// TwinCAT 3 PLC project Example
// ProgramVersion: 3.1.4024.0
// libraries:
//   MTP, * (Zerlauth)
//   Tc2_MC2, * (Beckhoff Automation GmbH)
//   Tc2_Standard, * (Beckhoff Automation GmbH)
//   Tc2_System, * (Beckhoff Automation GmbH)
//   Tc2_Utilities, * (Beckhoff Automation GmbH)
//   Tc3_Module, * (Beckhoff Automation GmbH)
// project tree:
//   GVLs/ GVL.TcGVL
//   / plcTask1.TcTTO
//   POUs/Axis/ FB_McAxis.TcPOU, I_Axis.TcIO
//   POUs/ FB_Alarm.TcPOU, FB_Module01.TcPOU, MAIN.TcPOU
// real-time tasks:
//   TASK plcTask1: cycle T#1000ms, priority 20, ADS port 350

CONFIGURATION Example
    RESOURCE PLC ON TwinCAT3
        TASK plcTask1(INTERVAL := T#1000ms, PRIORITY := 20);
        PROGRAM Task1 WITH plcTask1 : Task1;
    END_RESOURCE
END_CONFIGURATION

// ---- GVLs/GVL.TcGVL
VAR_GLOBAL
	fbSaftey:		FB_Component;	
END_VAR

// ---- POUs/Axis/I_Axis.TcIO
INTERFACE I_Axis

END_INTERFACE

// ---- POUs/Axis/FB_McAxis.TcPOU
FUNCTION_BLOCK FB_McAxis EXTENDS FB_Component IMPLEMENTS I_Axis
VAR_INPUT
	bHome:				BOOL;
END_VAR
VAR_OUTPUT
END_VAR
VAR
	// Structs
	stAxis:							AXIS_REF;
	stParameter:					ST_AxisParameterSet;
	stComponents:					ST_AxisComponents;
	
	// General
	fbPower: 						MC_Power;
	fbReset: 						MC_Reset;
	fbHome: 						MC_Home;

	// Motion function blocks
	fbJog:							MC_Jog;
	fbSetPosition: 					MC_SetPosition;
	fbMoveAbsolute: 				REFERENCE TO MC_MoveAbsolute := fbMoveAbsolute1;
	fbMoveAbsolute1: 				MC_MoveAbsolute;
	fbMoveAbsolute2: 				MC_MoveAbsolute;
	fbMoveVelocity: 				MC_MoveVelocity;
	fbMoveRelative: 				MC_MoveRelative;
	fbHalt: 						MC_Halt;
	fbStop: 						MC_Stop;
	
	// Read function blocks
	fbReadAxisComponents:			MC_ReadAxisComponents;	
	fbReadError: 					MC_ReadAxisError;
	fbReadParameterSet:				MC_ReadParameterSet;	
	fbReadBoolParameter:			MC_ReadBoolParameter;
	fbReadParameter: 				MC_ReadParameter;
	
	// Write function blocks                            		
	fbWriteBoolParameter: 			MC_WriteBoolParameter;
	fbWriteBoolParameterPersistent: MC_WriteBoolParameterPersistent;
	fbWriteParameter: 				MC_WriteParameter;
	fbWriteParameterPersistent: 	MC_WriteParameterPersistent;
END_VAR
VAR PERSISTENT
	bCalibration:					BOOL;
	fHomePosition:					LREAL;
	fPositionCorrection:			LREAL;
	fMaximumForce:					LREAL;
END_VAR


SUPER^();

stAxis.ReadStatus();

fbPower(Axis:= stAxis);
	
fbReset(Axis:= stAxis);
fbReset.Execute:= FALSE;

fbJog(Axis:= stAxis);
fbJog.JogForward:= FALSE;
fbJog.JogBackwards:= FALSE;

fbHome(Axis:= stAxis);
fbHome.Execute:= FALSE;
	
fbSetPosition(Axis:= stAxis);
fbSetPosition.Execute:= FALSE;

fbMoveAbsolute1(Axis:= stAxis);
fbMoveAbsolute1.Execute:= FALSE;
	
fbMoveAbsolute2(Axis:= stAxis);
fbMoveAbsolute2.Execute:= FALSE;
	
fbMoveRelative(Axis:= stAxis);
fbMoveRelative.Execute:= FALSE;
	
fbMoveVelocity(Axis:= stAxis);
fbMoveVelocity.Execute:= FALSE;

fbHalt(Axis:= stAxis);
fbHalt.Execute:= FALSE;
	
fbStop(Axis:= stAxis);
fbStop.Execute:= FALSE;
	
fbReadBoolParameter(Axis:= stAxis);
fbReadBoolParameter.Enable:= FALSE;

fbWriteBoolParameter(Axis:= stAxis);
fbWriteBoolParameter.Execute:= FALSE;

fbWriteBoolParameterPersistent(Axis:= stAxis);
fbWriteBoolParameterPersistent.Execute:= FALSE;

fbReadParameter(Axis:= stAxis);
fbReadParameter.Enable:= FALSE;
	
fbWriteParameter(Axis:= stAxis);
fbWriteParameter.Execute:= FALSE;

fbWriteParameterPersistent(Axis:= stAxis);
fbWriteParameterPersistent.Execute:= FALSE;
	
fbReadParameterSet(Parameter:=stParameter, Axis:= stAxis);
fbReadParameterSet.Execute:= FALSE;

fbReadAxisComponents(AxisComponents:= stComponents, Axis:= stAxis);
fbReadError(Axis:= stAxis, Enable:= TRUE);

IF stAxis.Status.NcApplicationRequest THEN
	M_Home(stParameter.fEncRefPosition, MC_HomingMode.MC_Direct, TRUE);
END_IF

stAxis.PlcToNc.PositionCorrection:= fPositionCorrection;

METHOD M_Calibration : BOOL
VAR_INPUT
	fPrePosition:	LREAL;
	fPosition:		LREAL;
	fForce:			LREAL;
	fLimit:			LREAL;
	bEvaluation:	BOOL;
END_VAR
VAR_OUTPUT
	fDeviation:		LREAL;
END_VAR
END_METHOD

METHOD PUBLIC M_Halt : BOOL
VAR_INPUT
END_VAR
fbHalt.Execute:= TRUE;
M_Halt:= stAxis.Status.NotMoving;
END_METHOD

METHOD PUBLIC M_Home : BOOL
VAR_INPUT
	fPosition:					LREAL;
	eHomingMode:				MC_HomingMode;
	bClearPositionLag: 			BOOL;
END_VAR
fbHome.Execute:= TRUE;
fbHome.Position:= fPosition;
fbHome.HomingMode:= eHomingMode;
fbHome.Options.ClearPositionLag:= bClearPositionLag;
IF fbHome.Done THEN
	fbReset.Execute:= TRUE;
	M_Home:= TRUE;
END_IF
END_METHOD

METHOD PUBLIC M_Jog : BOOL
VAR_INPUT
	bPositive:	BOOL;
	bNegative:	BOOL;
	eMode:		E_JogMode;
END_VAR
fbJog.Mode:= eMode;
IF bPositive AND NOT bNegative THEN
	fbJog.JogForward:= TRUE;
ELSIF bNegative AND NOT bPositive THEN
	fbJog.JogBackwards:= TRUE;
END_IF
M_Jog:= fbJog.Active;
END_METHOD

METHOD PUBLIC M_MoveAbsolute : BOOL
VAR_INPUT
	fPosition:				LREAL;
	fVelocity:				LREAL;
	fAcceleration:			LREAL;
	fDeceleration:			LREAL;
	fJerk:					LREAL;	
END_VAR
// Axis redy?
IF stAxis.Status.ControlLoopClosed THEN
	// input changed?
	IF fPosition <> fbMoveAbsolute.Position OR_ELSE fVelocity <> fbMoveAbsolute.Velocity OR_ELSE fbMoveAbsolute.Acceleration <> fbMoveAbsolute.Acceleration OR_ELSE fDeceleration <> fbMoveAbsolute.Deceleration OR_ELSE fJerk <> fbMoveAbsolute.Jerk THEN
		IF NOT fbMoveAbsolute1.Busy THEN
			// select axis 1
			fbMoveAbsolute:= fbMoveAbsolute1;
		ELSIF NOT fbMoveAbsolute2.Busy THEN
			// select axis 2
			fbMoveAbsolute:= fbMoveAbsolute2;
		ELSE
			// command blocked
			M_MoveAbsolute:= FALSE;
			RETURN;
		END_IF
		// take values
		fbMoveAbsolute.Execute:= 		TRUE;
		fbMoveAbsolute.Position:= 		fPosition;
		fbMoveAbsolute.Velocity:= 		fVelocity;
		fbMoveAbsolute.Acceleration:= 	fAcceleration;
		fbMoveAbsolute.Deceleration:= 	fDeceleration;
		fbMoveAbsolute.Jerk:= 			fJerk;
		M_MoveAbsolute:= FALSE;
	ELSE
		// Done
		M_MoveAbsolute:= stAxis.Status.InTargetPosition;
	END_IF
ELSE
	M_MoveAbsolute:= FALSE;
END_IF
END_METHOD

METHOD PUBLIC M_MoveRelative : BOOL
VAR_INPUT
	fDistance:				LREAL;
	fVelocity:				LREAL;
	fAcceleration:			LREAL;
	fDeceleration:			LREAL;
	fJerk:					LREAL;	
END_VAR
IF fbPower.Status THEN
	fbMoveRelative.Execute:= 			TRUE;
	fbMoveRelative.Distance:= 			fDistance;
	fbMoveRelative.Velocity:= 			fVelocity;
	fbMoveRelative.Acceleration:= 		fAcceleration;
	fbMoveRelative.Deceleration:= 		fDeceleration;
	fbMoveRelative.Jerk:= 				fJerk;
	M_MoveRelative:= 					fbMoveRelative.Done;
END_IF
END_METHOD

METHOD PUBLIC M_MoveVelocity : BOOL
VAR_INPUT
	fVelocity:				LREAL;
	fAcceleration:			LREAL;
	fDeceleration:			LREAL;
	fJerk:					LREAL;	
END_VAR
IF fbPower.Status THEN
	fbMoveVelocity.Execute:= 			TRUE;
	fbMoveVelocity.Velocity:= 			fVelocity;
	fbMoveVelocity.Acceleration:= 		fAcceleration;
	fbMoveVelocity.Deceleration:= 		fDeceleration;
	fbMoveVelocity.Jerk:= 				fJerk;
	IF fVelocity >= 0.0 THEN
		fbMoveVelocity.Direction:= 			MC_Direction.MC_Positive_Direction;
	ELSE
		fbMoveVelocity.Direction:= 			MC_Direction.MC_Negative_Direction;	
	END_IF
	
	M_MoveVelocity:= fbMoveVelocity.InVelocity;
END_IF
END_METHOD

METHOD PUBLIC M_PositionCorrection : BOOL
VAR_INPUT
	fPositionCorrection:		LREAL;
END_VAR
IF stAxis.Status.ControlLoopClosed THEN
	fbPower.Enable:= FALSE;
ELSE
	fbPower.Enable:= TRUE;
	fPositionCorrection:= fPositionCorrection;
	M_PositionCorrection:= stAxis.Status.ControlLoopClosed;
END_IF
END_METHOD

METHOD PUBLIC M_Power : BOOL
VAR_INPUT
	bOnOff:			BOOL;
END_VAR
IF bOnOff THEN
	fbReset.Execute:= TRUE;
	fbPower.Enable:= TRUE;
	fbPower.Enable_Negative:= TRUE;
	fbPower.Enable_Positive:= TRUE;
	fbPower.Override:= 100.0;
	fbPower.BufferMode:= MC_BufferMode.MC_Aborting;
	M_ReadParameterSet();
	M_ReadComponents();
	M_Power:= stAxis.Status.ControlLoopClosed;
ELSE
	fbPower.Enable:= FALSE;
	M_Power:= NOT stAxis.Status.ControlLoopClosed;
END_IF
END_METHOD

METHOD PUBLIC M_ReadBOOL : BOOL
VAR_INPUT
	 eParameterNumber:		MC_AxisParameter;		// MC_AxisParameter
	 bValue:				REFERENCE TO BOOL;
END_VAR
fbReadBoolParameter.Enable:= TRUE;
fbReadBoolParameter.ParameterNumber:= eParameterNumber;
fbReadBoolParameter.ReadMode:= E_ReadMode.READMODE_ONCE;
IF fbReadBoolParameter.Valid THEN
	IF __ISVALIDREF(bValue) THEN
		bValue:= fbReadBoolParameter.Value;
		M_ReadBOOL:= TRUE;		
	END_IF
END_IF
END_METHOD

METHOD PUBLIC M_ReadComponents : BOOL
VAR_INPUT
END_VAR
fbReadAxisComponents.Execute:= TRUE;
M_ReadComponents:= fbReadAxisComponents.Done;
END_METHOD

METHOD PUBLIC M_ReadLREAL : BOOL
VAR_INPUT
	 eParameterNumber:		MC_AxisParameter;		// MC_AxisParameter
	 fValue:				REFERENCE TO LREAL;
END_VAR
fbReadParameter.Enable:= TRUE;
fbReadParameter.ParameterNumber:= eParameterNumber;
fbReadParameter.ReadMode:= E_ReadMode.READMODE_ONCE;
IF fbReadParameter.Valid THEN
	IF __ISVALIDREF(fValue) THEN
		fValue:= fbReadParameter.Value;
		M_ReadLREAL:= TRUE;	
	END_IF
END_IF
END_METHOD

METHOD PUBLIC M_ReadParameterSet : BOOL
VAR_INPUT
END_VAR
fbReadParameterSet.Execute:= TRUE;
M_ReadParameterSet:= fbReadParameterSet.Done;
END_METHOD

METHOD PUBLIC M_Reset : BOOL
VAR_INPUT
END_VAR
fbReset.Execute:= TRUE;		
M_Reset:= fbReset.Done;
END_METHOD

METHOD PUBLIC M_SetPosition : BOOL
VAR_INPUT
	fPosition:					LREAL;
	bClearPositionLag: 			BOOL;
END_VAR
fbSetPosition.Execute:= TRUE;
fbSetPosition.Position:= fPosition;
fbSetPosition.Options.ClearPositionLag:= bClearPositionLag;
M_SetPosition:= fbSetPosition.Done;
END_METHOD

METHOD PUBLIC M_Stop : BOOL
VAR_INPUT
END_VAR
fbStop.Execute:= TRUE;
M_Stop:=  stAxis.Status.NotMoving;
END_METHOD

METHOD PUBLIC M_WriteBOOL : BOOL
VAR_INPUT
	eParameterNumber:		MC_AxisParameter;		// MC_AxisParameter
	bPersistent:			BOOL;
	bValue:					BOOL;
END_VAR
IF bPersistent THEN
	fbWriteBoolParameterPersistent.Execute:= TRUE;
	fbWriteBoolParameterPersistent.ParameterNumber:= eParameterNumber;
	fbWriteBoolParameterPersistent.Value:= bValue;
	IF fbWriteBoolParameterPersistent.Done THEN
		M_WriteBOOL:= TRUE;
	END_IF
ELSE
	fbWriteBoolParameter.Execute:= TRUE;
	fbWriteBoolParameter.ParameterNumber:= eParameterNumber;
	fbWriteBoolParameter.Value:= bValue;
	IF fbWriteBoolParameter.Done THEN
		M_WriteBOOL:= TRUE;
	END_IF
END_IF
END_METHOD

METHOD PUBLIC M_WriteLREAL : BOOL
VAR_INPUT
	eParameterNumber:		MC_AxisParameter;		// MC_AxisParameter
	bPersistent:			BOOL;
	fValue:					LREAL;
END_VAR
IF bPersistent THEN
	fbWriteParameterPersistent.Execute:= TRUE;
	fbWriteParameterPersistent.ParameterNumber:= eParameterNumber;
	fbWriteParameterPersistent.Value:= fValue;
	IF fbWriteParameterPersistent.Done THEN
		M_WriteLREAL:= TRUE;
	END_IF
ELSE
	fbWriteParameter.Execute:= TRUE;
	fbWriteParameter.ParameterNumber:= eParameterNumber;
	fbWriteParameter.Value:= fValue;
	IF fbWriteparameter.Done THEN
		M_WriteLREAL:= TRUE;
	END_IF
END_IF
END_METHOD

PROPERTY PUBLIC P_State : REFERENCE TO AXIS_REF
GET
P_State ref= stAxis;
END_GET
END_PROPERTY

END_FUNCTION_BLOCK

// ---- POUs/FB_Alarm.TcPOU
FUNCTION_BLOCK FB_Alarm IMPLEMENTS I_Logger
VAR_INPUT
END_VAR
VAR_OUTPUT
END_VAR
VAR
	nLength:		INT;
	aEvent:			ARRAY [0..nMax] OF ST_Event;
END_VAR
VAR CONSTANT
	nMax:			INT:= 99;
END_VAR

METHOD M_Find : DINT
VAR_INPUT
	stEvent	: 		ST_Event;
END_VAR
VAR
	nIndex: 	DINT;
END_VAR
// Object already in List
M_Find := -1;
WHILE nIndex < nLength DO
    IF (aEvent[nIndex].Source = stEvent.Source) 
		AND_THEN (aEvent[nIndex].EventType = stEvent.EventType) 
		AND_THEN (aEvent[nIndex].Message = stEvent.Message) THEN
			M_Find := nIndex;
			RETURN;
    END_IF
	nIndex := nIndex + 1;
END_WHILE
END_METHOD

METHOD M_Log
VAR_INPUT
	stEvent	: 		ST_Event;
END_VAR

VAR
	nIndex: DINT;
END_VAR
IF (nIndex:= M_Find(stEvent)) = -1 THEN
	aEvent[nLength]:= stEvent;
	nLength:= nLength + 1;
ELSE
	aEvent[nIndex]:= stEvent;	
END_IF
END_METHOD

END_FUNCTION_BLOCK

// ---- POUs/FB_Module01.TcPOU
FUNCTION_BLOCK FB_Module01 EXTENDS FB_Component
VAR_INPUT
END_VAR
VAR_OUTPUT
END_VAR
VAR
	fbLogger:					FB_ListLogger;
	fbAlarm:					FB_Alarm;
	fbComponent1:				FB_Component;
	fbComponent2:				FB_Component;
	fbComponent3:				FB_Component;
	fbComponent4:				FB_Component;
	bEvent: 					BOOL;
END_VAR

SUPER^();

fbComponent1();
fbComponent2();
fbComponent3();
fbComponent4();

IF bEvent THEN
	bEvent:= FALSE;
	fbComponent1.fbEvent.M_Add('Test');
	fbComponent1.fbEvent.M_Add('Test2');
	fbComponent1.fbEvent.M_Add('Test3');
	fbComponent1.fbEvent.M_Abort('First Error Abort',1);
END_IF

METHOD PROTECTED M_Initialise : BOOL
VAR_INPUT
END_VAR
IF SUPER^.M_Initialise() THEN
	fbLogger.M_Add(fbAlarm);

	fbSaftey.fbEvent.P_Logger:= fbLogger;
	fbSaftey.fbObserver.M_Attach(THIS^);


	fbComponent1.fbEvent.P_Logger:= fbLogger;
	fbComponent1.fbObserver.M_Attach(THIS^);
	fbObserver.M_Attach(fbComponent1);
	
	fbComponent2.fbEvent.P_Logger:= fbLogger;
	fbComponent2.fbObserver.M_Attach(THIS^);
	fbObserver.M_Attach(fbComponent2);
	
	fbComponent3.fbEvent.P_Logger:= fbLogger;
	fbComponent3.fbObserver.M_Attach(THIS^);
	fbObserver.M_Attach(fbComponent3);
	
	fbComponent4.fbEvent.P_Logger:= fbLogger;
	fbComponent4.fbObserver.M_Attach(THIS^);
	fbObserver.M_Attach(fbComponent4);
	M_Initialise:= TRUE;
END_IF
END_METHOD

METHOD PROTECTED M_Resetting : BOOL
VAR_INPUT
END_VAR
VAR
	nIndex:					DINT;
END_VAR
M_Resetting:= TRUE;
WHILE nIndex < fbObserver.nLength DO
	fbObserver.M_Index(nIndex).M_Request(E_Request.Reset);
	nIndex:= nIndex +1;
END_WHILE
END_METHOD

METHOD PROTECTED M_Starting : BOOL
VAR_INPUT
END_VAR
VAR
	nIndex:					DINT;
END_VAR
M_Starting:= TRUE;
WHILE nIndex < fbObserver.nLength DO
	M_Starting:= M_Starting AND fbObserver.M_Index(nIndex).M_Request(E_Request.Start);
	nIndex:= nIndex +1;
END_WHILE
END_METHOD

END_FUNCTION_BLOCK

// ---- POUs/MAIN.TcPOU
PROGRAM MAIN
VAR
	fbModule:		FB_Module01;	
	bReset:			BOOL;
	bStart: 		BOOL;
    bHold:       	BOOL;
    bPause:    		BOOL;
	bStop:       	BOOL;
    bAbort:      	BOOL;

END_VAR


fbSaftey();
fbModule();

IF bReset THEN
	bReset:= NOT fbModule.M_Request(E_Request.Reset);
END_IF

IF bStart THEN
	bStart:= NOT fbModule.M_Request(E_Request.Start);
END_IF

IF bStop THEN
	bStop:= fbModule.M_Request(E_Request.Stop);
END_IF

IF bHold THEN
	bHold:= NOT fbModule.M_Request(E_Request.Hold);
END_IF

IF bPause THEN
	bPause:= NOT fbModule.M_Request(E_Request.Pause);
END_IF

IF bAbort THEN
	bAbort:= NOT fbModule.M_Request(E_Request.Abort);
END_IF

END_PROGRAM
